{attribute 'qualified_only'}
VAR_GLOBAL
END_VAR
VAR_GLOBAL CONSTANT
    MAX_RELATED_GROUPS : USINT := 19;
END_VAR

(* stored: Version 1.1.0.1
   GVL GVLTcCommando: Id {1c792e27-feb4-0b48-1cf6-c8147134d538} *)
